{attribute 'GeneratedUsingTerminal: EL3403-0000-0018'}
{attribute addProperty BoxType "EL3403-0000-0018"}
{attribute addProperty Description "EL3403 3Ch. Power Measuring"}
{attribute addProperty Physics "KK"}
{attribute addProperty Id "PM_Inputs_Channel_1AT %I*PM_Inputs_Channel_2468BF1D19PM_Inputs_Channel_2AT %I*PM_Inputs_Channel_2468BF1D19PM_Inputs_Channel_3AT %I*PM_Inputs_Channel_2468BF1D19PM_Status_dataAT %I*PM_Status_data_0FD072A05PM_Outputs_Channel_1AT %Q*PM_Outputs_Channel_E5FBDE301PM_Outputs_Channel_2AT %Q*PM_Outputs_Channel_E5FBDE301PM_Outputs_Channel_3AT %Q*PM_Outputs_Channel_E5FBDE301WcStateAT %I*WcState_9091E0EB2InfoDataAT %I*InfoData_32EB74EA10"}
{attribute addProperty CRC "3040281115"}
{attribute addProperty Size "77"}
TYPE EL3403_B537021B EXTENDS EtcSlaveTerminalBase_947E5A46 :
STRUCT
	{attribute addProperty Name "PM_Inputs_Channel_1"}
	PM_Inputs_Channel_1 : PM_Inputs_Channel_2468BF1D;
	{attribute addProperty Name "PM_Inputs_Channel_2"}
	PM_Inputs_Channel_2 : PM_Inputs_Channel_2468BF1D;
	{attribute addProperty Name "PM_Inputs_Channel_3"}
	PM_Inputs_Channel_3 : PM_Inputs_Channel_2468BF1D;
	{attribute addProperty Name "PM_Status_data"}
	PM_Status_data : PM_Status_data_0FD072A0;
	{attribute addProperty Name "PM_Outputs_Channel_1"}
	PM_Outputs_Channel_1 : PM_Outputs_Channel_E5FBDE30;
	{attribute addProperty Name "PM_Outputs_Channel_2"}
	PM_Outputs_Channel_2 : PM_Outputs_Channel_E5FBDE30;
	{attribute addProperty Name "PM_Outputs_Channel_3"}
	PM_Outputs_Channel_3 : PM_Outputs_Channel_E5FBDE30;
	{attribute addProperty Name "WcState"}
	WcState : WcState_9091E0EB;
	{attribute addProperty Name "InfoData"}
	InfoData : InfoData_32EB74EA;
END_STRUCT
END_TYPE

(* stored: Version 1.2.0.0, ProductVersion 3.1.4024.11
   DUT EL3403_B537021B: Id {e97012a5-a49a-463b-acb8-56228a284c39} *)
